FUNCTION_BLOCK Person Extends Object
VAR_INPUT
END_VAR
VAR_OUTPUT
END_VAR
VAR
    _age : INT;
    _name : STRING;
END_VAR

METHOD Equals : BOOL
VAR_INPUT
    other : I_Equatable;
END_VAR
IF GetAge() = GVL.CastHelper.I_EquatableToPerson(other)^.GetAge() THEN
    Equals := TRUE;
ELSE
    Equals := FALSE;
END_IF
END_METHOD

METHOD GetAge : int
VAR_INPUT
END_VAR
GetAge := _age;
END_METHOD

METHOD PUBLIC GetName : STRING
GetName := _name;
END_METHOD

METHOD SetAge : int
VAR_INPUT
    age : int;
END_VAR
_age := age;
SetAge := _age;
END_METHOD

METHOD PUBLIC SetName : STRING
VAR_INPUT
    name : STRING;
END_VAR
_name := name;
SetName := _name;
END_METHOD

END_FUNCTION_BLOCK

(* stored: Version 1.1.0.1, ProductVersion 3.1.4024.6
   POU Person: Id {b35078b8-f2ca-46dd-b46c-a75c80a795cc}, SpecialFunc None
   Method Equals: Id {11e1f2c0-8e08-4a87-b65f-5107d7629633}
   Method GetAge: Id {de6e54a3-dee1-429d-98ce-448ad1488ce6}
   Method GetName: Id {e4d9f3f5-7f81-46fa-abcb-51aadbd75627}
   Method SetAge: Id {9a4bd406-b6ed-42f8-b11a-3f8c9068e4d4}
   Method SetName: Id {28bf7cbf-f50a-4e9c-8e76-c1bc7c107c08} *)
